// TIA Portal V19 export
FUNCTION_BLOCK "A0303_Sostegno_FB"   // FB102, LAD
// stored: MemoryReserve 100, SetENOAutomatically false
   VAR_INPUT
      AreaInterface : "AreaInterface";
      ZSI : "udt_ZoneSafetyInterface";
      DSI_Feed : "udt_DeviceSafetyInterface";
      DSI_Valve : "udt_DeviceSafetyInterface";
      DataIn : Struct
         OP_Work_PB : Bool;
         OP_Rest_PB : Bool;
         Pos0_Ls : Bool;
         Pos1_Ls : Bool;
         Pos2_Ls : Bool;
      END_STRUCT;
      CIn : Struct
         Manager : Struct
            EnableStopDoorOpeningReq : Bool;
            EnableStopInPhase : Bool;
            EnableStopProgrammed : Bool;
            Control_ON : Bool;
            CanMoveFreely : Bool;
            Phase : Struct
               VAI_A_LAVORO : Bool;
               VAI_A_RIPOSO : Bool;
            END_STRUCT;
            Ax : Struct
               Pos { ExternalVisible := 'False'; ExternalWritable := 'False'} : LReal;
            END_STRUCT;
            Paletti : Struct
               PosPaletto : Int;
               Pos1Collision : Bool;
               Pos2Collision : Bool;
            END_STRUCT;
         END_STRUCT;
         Navetta : Struct
            OutOfWorkspace : Bool;
         END_STRUCT;
         Trasporto : Struct
            OutOfWorkspace : Bool;
         END_STRUCT;
         CycleModeShortPiece : Bool;
      END_STRUCT;
      Config : Struct
         Ax : "Positioning_DOL_Machine_Config";
         V_1 : "ValveMachine_Config";
         V_2 : "ValveMachine_Config";
         DelayMissingCondition { ExternalAccessible := 'False'; ExternalVisible := 'False'; ExternalWritable := 'False'} : Time;
      END_STRUCT;
      HWID : Struct
         Ax_TEL1 : HW_SUBMODULE;
         Enc_IO : HW_SUBMODULE;
      END_STRUCT;
   END_VAR
   VAR_OUTPUT
      MachineInterface : "MachineInterface";
      COut : Struct
         Ax : "Positioning_DOL_Machine_COut";
         Paletto : Struct
            CtrlSafe : Bool;
            Standstill : Bool;
            Rest_CheckNext : Bool;
            Work_CheckNext : Bool;
            Pos : Int;
            RestPosition : Bool;
         END_STRUCT;
      END_STRUCT;
   END_VAR
   VAR_IN_OUT
      Par : Struct
         Ax : "Positioning_DOL_Machine_Par";
         Ax_Pers : "Positioning_DOL_Machine_Pers_Data";
         Enc : "PosFbk_RTN";
      END_STRUCT;
      Par_Mach : Struct
         RestPosition : LReal;
         ToleranceWindow : LReal;
         PosTimeout : Time;
      END_STRUCT;
   END_VAR
   VAR
      Alarm : Struct
         Ax { S7_SetPoint := 'True'} : "Positioning_DOL_Machine_Alr";
         V_1 : "ValveAlr";
         V_2 : "ValveAlr";
         Enc { S7_SetPoint := 'True'} : "PosFbk_Encoder_Alr";
         Missing_Pos0_Ls_ON { S7_SetPoint := 'True'} : Bool;
         Missing_Pos1_Ls_ON { S7_SetPoint := 'True'} : Bool;
         Missing_Pos2_Ls_ON { S7_SetPoint := 'True'} : Bool;
         LimitSwitch : Bool;
      END_STRUCT;
      Warning : Struct
         Ax { S7_SetPoint := 'True'} : "Positioning_DOL_Machine_Wng";
         V_1 { S7_SetPoint := 'True'} : "ValveMachine_Wng";
         V_2 { S7_SetPoint := 'True'} : "ValveMachine_Wng";
         V_Paletti { S7_SetPoint := 'True'} : "ValveMachine_Wng";
         MissingCnd : Struct
            OP_REST : Bool;   // Mancanza comando arresto
            OP_WORK : Bool;   // Mancanza consenso lavoro
            AxInRestPos : Bool;
         END_STRUCT;
      END_STRUCT;
      Ctrl : Struct
         Man : Struct
            OP_Vai_A_Lavoro : Bool;
            OP_Vai_A_Riposo : Bool;
         END_STRUCT;
         Aut : Struct
            OP_Vai_A_Lavoro : Bool;
            OP_Vai_A_Riposo : Bool;
         END_STRUCT;
         Pos0 : Bool;
         Pos1 : Bool;
         Pos2 : Bool;
         OP_Vai_A_Lavoro : Bool;
         OP_Vai_A_Riposo : Bool;
      END_STRUCT;
      Sts : Struct
         OP_Ax_CanMoveFreely : Bool;
         OP_CanMoveFreely : Bool;
         OP_Rest_Cnd : Bool;
         OP_Work_Cnd : Bool;
         InRestPos : Bool;
      END_STRUCT;
      HMI : Struct
         PbPreset : Bool;
         PresetValue : LReal;
      END_STRUCT;
      Ax { S7_SetPoint := 'True'} : "Positioning_DOL_Machine_FB";
      Enc : "PosFbk_SickAFM60";
      Enc_ITF : "PosFbk_ITF";
      V_1 { S7_SetPoint := 'True'} : "ValveMachine_FB";
      V_2 { S7_SetPoint := 'True'} : "ValveMachine_FB";
      AUX : Struct
         OP_Work_PB { ExternalAccessible := 'False'; ExternalVisible := 'False'; ExternalWritable := 'False'} : Bool;
         OP_Rest_PB { ExternalAccessible := 'False'; ExternalVisible := 'False'; ExternalWritable := 'False'} : Bool;
         OP_MoveToPos : Bool;
         PbPos0 : Bool;
         PbPos1 : Bool;
         PbPos2 : Bool;
      END_STRUCT;
      TON_MissingLsPos0 : IEC_TIMER;
      TON_MissingLsPos1 : IEC_TIMER;
      TON_MissingLsPos2 : IEC_TIMER;
      TON_OP_REST_MissingCnd : IEC_TIMER;
      TON_OP_WORK_MissingCnd : IEC_TIMER;
   END_VAR
   VAR_TEMP
      PE : Struct
         OP_Rest_PB : Bool;
         OP_Work_PB : Bool;
         PbPos0 : Bool;
         PbPos1 : Bool;
         PbPos2 : Bool;
      END_STRUCT;
      V1_Work_1 : Bool;
      V1_Work_2 : Bool;
      V1_Rest : Bool;
      V1_Rest_2 : Bool;
      V2_Work : Bool;
      V2_Rest_1 : Bool;
      V2_Rest_2 : Bool;
   END_VAR
   VAR_TEMP   // added for the SCL form of the ladder/FBD networks
      _w1 : Bool;
   END_VAR
BEGIN

REGION Network 1 (SCL): Reset allarmi
   IF #AreaInterface.RstAlarms THEN
       #Warning.MissingCnd.AxInRestPos:=FALSE;
   END_IF;
END_REGION

REGION Network 2: <+>
END_REGION

REGION Network 3: <+>
END_REGION

REGION Network 4: [Ax] - Operazione può muoversi liberamente perchè non sposta nessun BEAM
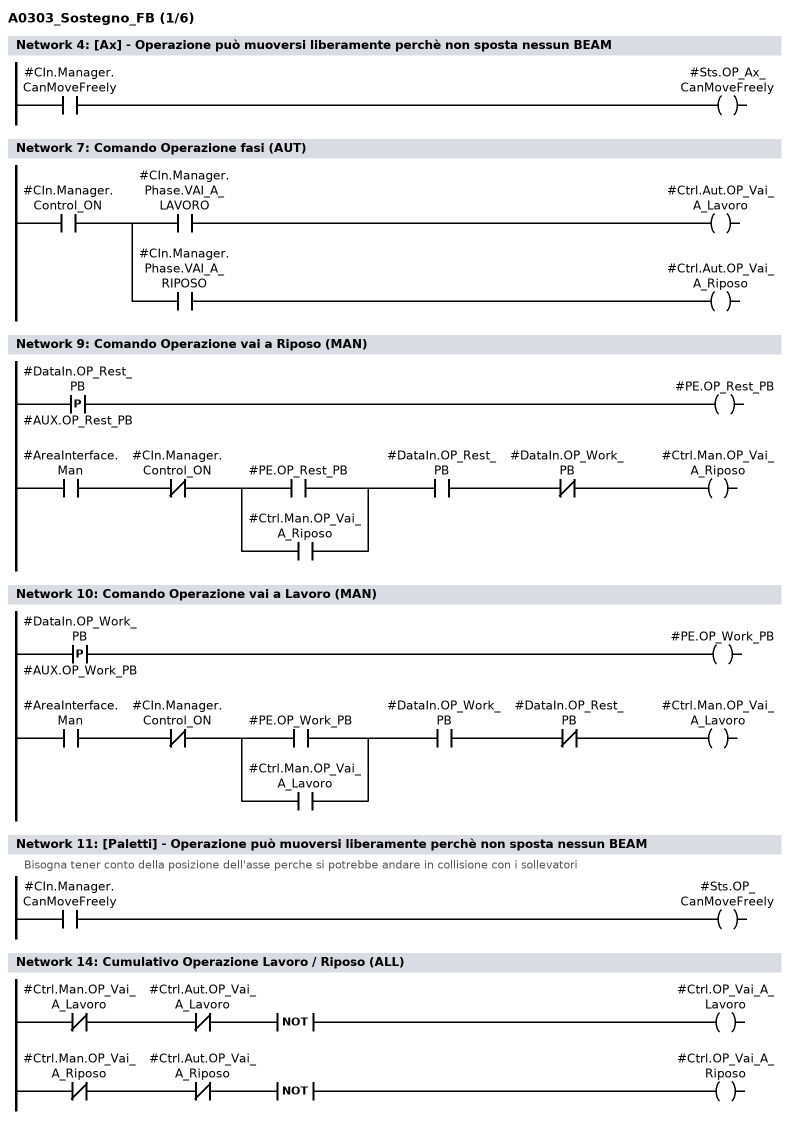
   RUNG wire#powerrail
      Contact( #CIn.Manager.CanMoveFreely )
      Coil( #Sts.OP_Ax_CanMoveFreely )
   END_RUNG
   // the same network as SCL:
   #Sts.OP_Ax_CanMoveFreely := #CIn.Manager.CanMoveFreely;
END_REGION

REGION Network 5: <+>
END_REGION

REGION Network 6: < OPERAZIONI AUTOMATICO >
END_REGION

REGION Network 7: Comando Operazione fasi (AUT)
   RUNG wire#powerrail
      Contact( #CIn.Manager.Control_ON )
      wire#w1
      Contact( #CIn.Manager.Phase.VAI_A_LAVORO )
      Coil( #Ctrl.Aut.OP_Vai_A_Lavoro )
   END_RUNG
   RUNG wire#w1
      Contact( #CIn.Manager.Phase.VAI_A_RIPOSO )
      Coil( #Ctrl.Aut.OP_Vai_A_Riposo )
   END_RUNG
   // the same network as SCL:
   #Ctrl.Aut.OP_Vai_A_Lavoro := #CIn.Manager.Control_ON AND #CIn.Manager.Phase.VAI_A_LAVORO;
   #Ctrl.Aut.OP_Vai_A_Riposo := #CIn.Manager.Control_ON AND #CIn.Manager.Phase.VAI_A_RIPOSO;
END_REGION

REGION Network 8: < OPERAZIONI MANUALI >
END_REGION

REGION Network 9: Comando Operazione vai a Riposo (MAN)
   RUNG wire#powerrail
      P_Contact(operand := #DataIn.OP_Rest_PB, bit := #AUX.OP_Rest_PB)
      Coil( #PE.OP_Rest_PB )
   END_RUNG
   RUNG wire#powerrail
      Contact( #AreaInterface.Man )
      I_Contact( #CIn.Manager.Control_ON )
      wire#w1
      Contact( #PE.OP_Rest_PB )
      wire#w2
      Contact( #DataIn.OP_Rest_PB )
      I_Contact( #DataIn.OP_Work_PB )
      Coil( #Ctrl.Man.OP_Vai_A_Riposo )
   END_RUNG
   RUNG wire#w1
      Contact( #Ctrl.Man.OP_Vai_A_Riposo )
   END_RUNG wire#w2
   // the same network as SCL:
   #_w1 := #DataIn.OP_Rest_PB AND NOT #AUX.OP_Rest_PB;   // rising edge of #DataIn.OP_Rest_PB
   #AUX.OP_Rest_PB := #DataIn.OP_Rest_PB;
   #PE.OP_Rest_PB := #_w1;
   #Ctrl.Man.OP_Vai_A_Riposo := #AreaInterface.Man AND NOT #CIn.Manager.Control_ON AND (#PE.OP_Rest_PB OR #Ctrl.Man.OP_Vai_A_Riposo) AND #DataIn.OP_Rest_PB AND NOT #DataIn.OP_Work_PB;
END_REGION

REGION Network 10: Comando Operazione vai a Lavoro (MAN)
   RUNG wire#powerrail
      P_Contact(operand := #DataIn.OP_Work_PB, bit := #AUX.OP_Work_PB)
      Coil( #PE.OP_Work_PB )
   END_RUNG
   RUNG wire#powerrail
      Contact( #AreaInterface.Man )
      I_Contact( #CIn.Manager.Control_ON )
      wire#w1
      Contact( #PE.OP_Work_PB )
      wire#w2
      Contact( #DataIn.OP_Work_PB )
      I_Contact( #DataIn.OP_Rest_PB )
      Coil( #Ctrl.Man.OP_Vai_A_Lavoro )
   END_RUNG
   RUNG wire#w1
      Contact( #Ctrl.Man.OP_Vai_A_Lavoro )
   END_RUNG wire#w2
   // the same network as SCL:
   #_w1 := #DataIn.OP_Work_PB AND NOT #AUX.OP_Work_PB;   // rising edge of #DataIn.OP_Work_PB
   #AUX.OP_Work_PB := #DataIn.OP_Work_PB;
   #PE.OP_Work_PB := #_w1;
   #Ctrl.Man.OP_Vai_A_Lavoro := #AreaInterface.Man AND NOT #CIn.Manager.Control_ON AND (#PE.OP_Work_PB OR #Ctrl.Man.OP_Vai_A_Lavoro) AND #DataIn.OP_Work_PB AND NOT #DataIn.OP_Rest_PB;
END_REGION

REGION Network 11: [Paletti] - Operazione può muoversi liberamente perchè non sposta nessun BEAM
   // Bisogna tener conto della posizione dell'asse perche si potrebbe andare in collisione con i sollevatori
   RUNG wire#powerrail
      Contact( #CIn.Manager.CanMoveFreely )
      Coil( #Sts.OP_CanMoveFreely )
   END_RUNG
   // the same network as SCL:
   #Sts.OP_CanMoveFreely := #CIn.Manager.CanMoveFreely;
END_REGION

REGION Network 12: <+>
END_REGION

REGION Network 13: < CUMULATIVO OPERAZIONI >
END_REGION

REGION Network 14: Cumulativo Operazione Lavoro / Riposo (ALL)
   RUNG wire#powerrail
      I_Contact( #Ctrl.Man.OP_Vai_A_Lavoro )
      I_Contact( #Ctrl.Aut.OP_Vai_A_Lavoro )
      Not()
      Coil( #Ctrl.OP_Vai_A_Lavoro )
   END_RUNG
   RUNG wire#powerrail
      I_Contact( #Ctrl.Man.OP_Vai_A_Riposo )
      I_Contact( #Ctrl.Aut.OP_Vai_A_Riposo )
      Not()
      Coil( #Ctrl.OP_Vai_A_Riposo )
   END_RUNG
   // the same network as SCL:
   #Ctrl.OP_Vai_A_Lavoro := NOT (NOT #Ctrl.Man.OP_Vai_A_Lavoro AND NOT #Ctrl.Aut.OP_Vai_A_Lavoro);
   #Ctrl.OP_Vai_A_Riposo := NOT (NOT #Ctrl.Man.OP_Vai_A_Riposo AND NOT #Ctrl.Aut.OP_Vai_A_Riposo);
END_REGION

REGION Network 15: < CONDIZIONI MOVIMENTO >
END_REGION

REGION Network 16: Condizioni movimento Operazione a Lavoro / Riposo
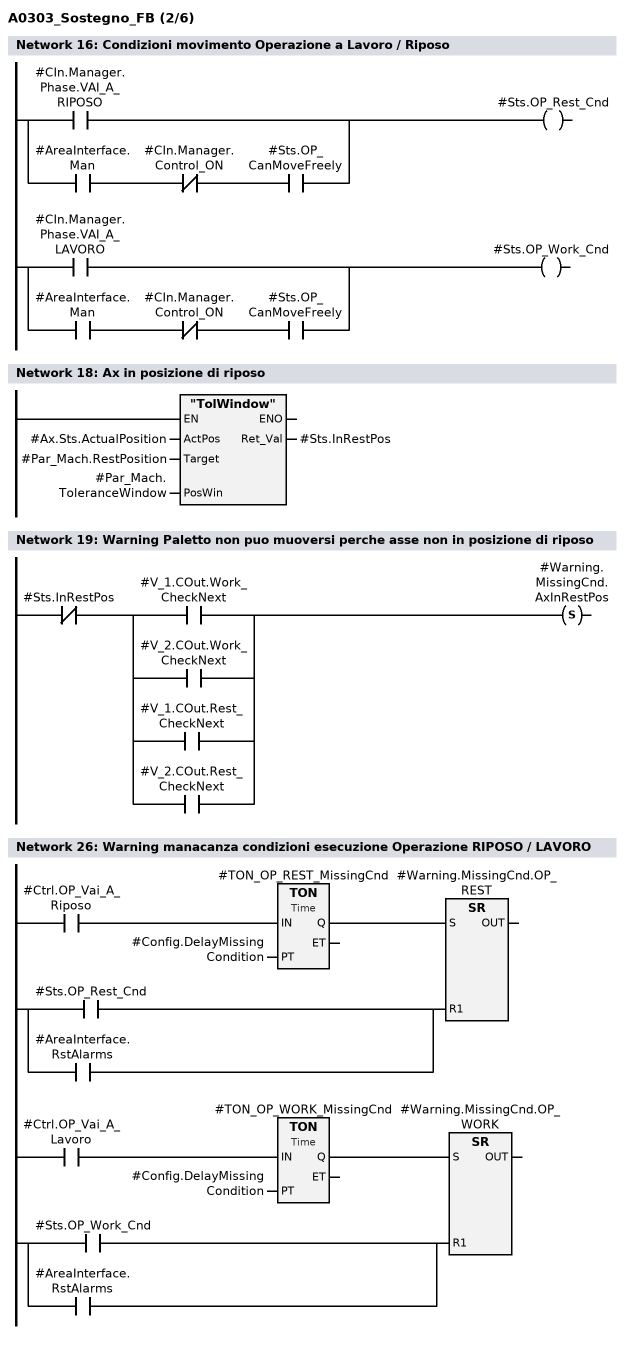
   RUNG wire#powerrail
      Contact( #CIn.Manager.Phase.VAI_A_RIPOSO )
      wire#w1
      Coil( #Sts.OP_Rest_Cnd )
   END_RUNG
   RUNG wire#powerrail
      Contact( #AreaInterface.Man )
      I_Contact( #CIn.Manager.Control_ON )
      Contact( #Sts.OP_CanMoveFreely )
   END_RUNG wire#w1
   RUNG wire#powerrail
      Contact( #CIn.Manager.Phase.VAI_A_LAVORO )
      wire#w2
      Coil( #Sts.OP_Work_Cnd )
   END_RUNG
   RUNG wire#powerrail
      Contact( #AreaInterface.Man )
      I_Contact( #CIn.Manager.Control_ON )
      Contact( #Sts.OP_CanMoveFreely )
   END_RUNG wire#w2
   // the same network as SCL:
   #Sts.OP_Rest_Cnd := #CIn.Manager.Phase.VAI_A_RIPOSO OR (#AreaInterface.Man AND NOT #CIn.Manager.Control_ON AND #Sts.OP_CanMoveFreely);
   #Sts.OP_Work_Cnd := #CIn.Manager.Phase.VAI_A_LAVORO OR (#AreaInterface.Man AND NOT #CIn.Manager.Control_ON AND #Sts.OP_CanMoveFreely);
END_REGION

REGION Network 17: <+>
END_REGION

REGION Network 18: Ax in posizione di riposo
   RUNG wire#powerrail
      "TolWindow"(ActPos := #Ax.Sts.ActualPosition, Target := #Par_Mach.RestPosition, PosWin := #Par_Mach.ToleranceWindow, Ret_Val => #Sts.InRestPos)
   END_RUNG
   // the same network as SCL:
   #Sts.InRestPos := "TolWindow"(ActPos := #Ax.Sts.ActualPosition,
                           Target := #Par_Mach.RestPosition,
                           PosWin := #Par_Mach.ToleranceWindow);
END_REGION

REGION Network 19: Warning Paletto non puo muoversi perche asse non in posizione di riposo
   RUNG wire#powerrail
      I_Contact( #Sts.InRestPos )
      wire#w1
      Contact( #V_1.COut.Work_CheckNext )
      wire#w2
      S_Coil( #Warning.MissingCnd.AxInRestPos )
   END_RUNG
   RUNG wire#w1
      Contact( #V_2.COut.Work_CheckNext )
   END_RUNG wire#w2
   RUNG wire#w1
      Contact( #V_1.COut.Rest_CheckNext )
   END_RUNG wire#w2
   RUNG wire#w1
      Contact( #V_2.COut.Rest_CheckNext )
   END_RUNG wire#w2
   // the same network as SCL:
   IF NOT #Sts.InRestPos AND (#V_1.COut.Work_CheckNext OR #V_2.COut.Work_CheckNext OR #V_1.COut.Rest_CheckNext OR #V_2.COut.Rest_CheckNext) THEN
       #Warning.MissingCnd.AxInRestPos := TRUE;
   END_IF;
END_REGION

REGION Network 20: <+>
END_REGION

REGION Network 21 (SCL): CIn Abilitazioni Manager
   //Stop Door Opening Request
   #Ax.CIn.Manager.EnableStopDoorOpeningReq :=
   #V_1.Cin.Manager.EnableStopDoorOpeningReq := #V_2.Cin.Manager.EnableStopDoorOpeningReq := #CIn.Manager.EnableStopDoorOpeningReq;

   //Stop In Phase
   #Ax.CIn.Manager.EnableStopInPhase := 
   #V_1.Cin.Manager.EnableStopInPhase := #V_2.Cin.Manager.EnableStopInPhase := #CIn.Manager.EnableStopInPhase;

   //Stop Programmed
   #Ax.CIn.Manager.EnableStopProgrammed := 
   #V_1.Cin.Manager.EnableStopProgrammed := #V_2.Cin.Manager.EnableStopProgrammed :=#CIn.Manager.EnableStopProgrammed;
END_REGION

REGION Network 22: <+>
END_REGION

REGION Network 23: <+>
END_REGION

REGION Network 24: <<<MANAGER >>>
END_REGION

REGION Network 25 (SCL): Cin Manager (Esecuzione sequenza comandi)
   //CTRL ON
   #Ax.CIn.Manager.Control_ON :=#V_1.Cin.Manager.Control_ON :=#V_2.Cin.Manager.Control_ON := #Ctrl.OP_Vai_A_Lavoro OR #Ctrl.OP_Vai_A_Riposo;


   IF #Ctrl.OP_Vai_A_Lavoro AND #Sts.OP_Work_Cnd THEN


       IF #CIn.Manager.Paletti.PosPaletto = 1 THEN
           #Ctrl.Pos1 := NOT #DataIn.Pos1_Ls;
       ELSIF #CIn.Manager.Paletti.PosPaletto = 2 THEN
           #Ctrl.Pos2 := NOT #DataIn.Pos2_Ls;
       END_IF;

       #Ax.CIn.Manager.Speed := 100;
       #Ax.CIn.Manager.MoveToPos := #CIn.Manager.Paletti.PosPaletto = #COut.Paletto.Pos;
       #Ax.CIn.Manager.Pos := #CIn.Manager.Ax.Pos;




   ELSIF #Ctrl.OP_Vai_A_Riposo AND #Sts.OP_Rest_Cnd THEN



       IF NOT #CIn.CycleModeShortPiece THEN

           #Ax.CIn.Manager.Speed := 100;
           #Ax.CIn.Manager.MoveToPos := #CIn.Manager.Paletti.PosPaletto = #COut.Paletto.Pos;
           #Ax.CIn.Manager.Pos := #Par_Mach.RestPosition;

           IF #Sts.InRestPos THEN
               #Ctrl.Pos0 := NOT #DataIn.Pos0_Ls;
           END_IF;

       ELSE

           #Ctrl.Pos0 := NOT #DataIn.Pos0_Ls;


       END_IF;

   ELSE
       #Ctrl.Pos0 := #Ctrl.Pos1 := #Ctrl.Pos2 :=  #Ax.CIn.Manager.MoveToPos:= FALSE;


   END_IF;
END_REGION

REGION Network 26: Warning manacanza condizioni esecuzione Operazione RIPOSO / LAVORO
   RUNG wire#powerrail
      Contact( #Ctrl.OP_Vai_A_Riposo )
      { S7_Templates := "time_type := Time" } #TON_OP_REST_MissingCnd.TON(pt := #Config.DelayMissingCondition, et =>)
      S_SR(operand := #Warning.MissingCnd.OP_REST, r1 := wire#w1)
   END_RUNG
   RUNG wire#powerrail
      Contact( #Sts.OP_Rest_Cnd )
   END_RUNG wire#w1
   RUNG wire#powerrail
      Contact( #AreaInterface.RstAlarms )
   END_RUNG wire#w1
   RUNG wire#powerrail
      Contact( #Ctrl.OP_Vai_A_Lavoro )
      { S7_Templates := "time_type := Time" } #TON_OP_WORK_MissingCnd.TON(pt := #Config.DelayMissingCondition, et =>)
      S_SR(operand := #Warning.MissingCnd.OP_WORK, r1 := wire#w2)
   END_RUNG
   RUNG wire#powerrail
      Contact( #Sts.OP_Work_Cnd )
   END_RUNG wire#w2
   RUNG wire#powerrail
      Contact( #AreaInterface.RstAlarms )
   END_RUNG wire#w2
   // the same network as SCL:
   #TON_OP_REST_MissingCnd.TON(IN := #Ctrl.OP_Vai_A_Riposo, PT := #Config.DelayMissingCondition);
   IF #TON_OP_REST_MissingCnd.Q THEN
       #Warning.MissingCnd.OP_REST := TRUE;   // SR flip-flop
   END_IF;
   IF #Sts.OP_Rest_Cnd OR #AreaInterface.RstAlarms THEN #Warning.MissingCnd.OP_REST := FALSE; END_IF;
   #TON_OP_WORK_MissingCnd.TON(IN := #Ctrl.OP_Vai_A_Lavoro, PT := #Config.DelayMissingCondition);
   IF #TON_OP_WORK_MissingCnd.Q THEN
       #Warning.MissingCnd.OP_WORK := TRUE;   // SR flip-flop
   END_IF;
   IF #Sts.OP_Work_Cnd OR #AreaInterface.RstAlarms THEN #Warning.MissingCnd.OP_WORK := FALSE; END_IF;
END_REGION

REGION Network 27: <+>
END_REGION

REGION Network 28: <<< ASSE Y >>>
END_REGION

REGION Network 29: [Ax] - Cin Ext Enable
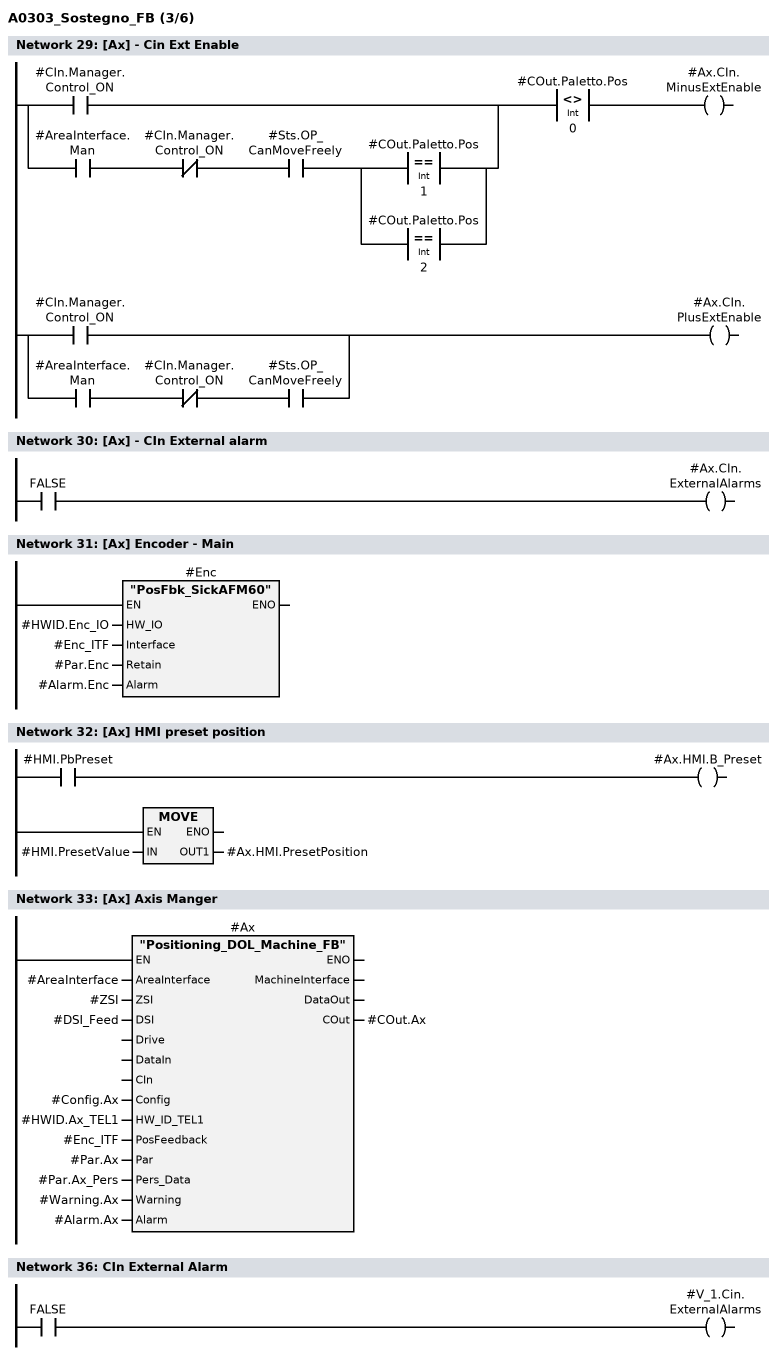
   RUNG wire#powerrail
      Contact( #CIn.Manager.Control_ON )
      wire#w1
      { S7_Templates := "SrcType := Int" } NE_Contact(in1 := #COut.Paletto.Pos, in2 := 0)
      Coil( #Ax.CIn.MinusExtEnable )
   END_RUNG
   RUNG wire#powerrail
      Contact( #AreaInterface.Man )
      I_Contact( #CIn.Manager.Control_ON )
      Contact( #Sts.OP_CanMoveFreely )
      wire#w2
      { S7_Templates := "SrcType := Int" } EQ_Contact(in1 := #COut.Paletto.Pos, in2 := 1)
   END_RUNG wire#w1
   RUNG wire#w2
      { S7_Templates := "SrcType := Int" } EQ_Contact(in1 := #COut.Paletto.Pos, in2 := 2)
   END_RUNG wire#w1
   RUNG wire#powerrail
      Contact( #CIn.Manager.Control_ON )
      wire#w3
      Coil( #Ax.CIn.PlusExtEnable )
   END_RUNG
   RUNG wire#powerrail
      Contact( #AreaInterface.Man )
      I_Contact( #CIn.Manager.Control_ON )
      Contact( #Sts.OP_CanMoveFreely )
   END_RUNG wire#w3
   // the same network as SCL:
   #Ax.CIn.MinusExtEnable := (#CIn.Manager.Control_ON OR (#AreaInterface.Man AND NOT #CIn.Manager.Control_ON AND #Sts.OP_CanMoveFreely AND ((#COut.Paletto.Pos = 1) OR (#COut.Paletto.Pos = 2)))) AND (#COut.Paletto.Pos <> 0);
   #Ax.CIn.PlusExtEnable := #CIn.Manager.Control_ON OR (#AreaInterface.Man AND NOT #CIn.Manager.Control_ON AND #Sts.OP_CanMoveFreely);
END_REGION

REGION Network 30: [Ax] - CIn External alarm
   RUNG wire#powerrail
      Contact( FALSE )
      Coil( #Ax.CIn.ExternalAlarms )
   END_RUNG
   // the same network as SCL:
   #Ax.CIn.ExternalAlarms := FALSE;
END_REGION

REGION Network 31: [Ax] Encoder - Main
   RUNG wire#powerrail
      #Enc(HW_IO := #HWID.Enc_IO, Interface := #Enc_ITF, Retain := #Par.Enc, Alarm := #Alarm.Enc)
   END_RUNG
   // the same network as SCL:
   #Enc(HW_IO := #HWID.Enc_IO, Interface := #Enc_ITF, Retain := #Par.Enc, Alarm := #Alarm.Enc);   // "PosFbk_SickAFM60"
END_REGION

REGION Network 32: [Ax] HMI preset position
   RUNG wire#powerrail
      Contact( #HMI.PbPreset )
      Coil( #Ax.HMI.B_Preset )
   END_RUNG
   RUNG wire#powerrail
      Move(in := #HMI.PresetValue, out1 => #Ax.HMI.PresetPosition)
   END_RUNG
   // the same network as SCL:
   #Ax.HMI.B_Preset := #HMI.PbPreset;
   #Ax.HMI.PresetPosition := #HMI.PresetValue;
END_REGION

REGION Network 33: [Ax] Axis Manger
   RUNG wire#powerrail
      #Ax(AreaInterface := #AreaInterface, ZSI := #ZSI, DSI := #DSI_Feed, Drive :=, DataIn :=, CIn :=, Config := #Config.Ax, HW_ID_TEL1 := #HWID.Ax_TEL1, PosFeedback := #Enc_ITF, Par := #Par.Ax, Pers_Data := #Par.Ax_Pers, Warning := #Warning.Ax, Alarm := #Alarm.Ax, MachineInterface =>, DataOut =>, COut => #COut.Ax)
   END_RUNG
   // the same network as SCL:
   #Ax(AreaInterface := #AreaInterface,   // "Positioning_DOL_Machine_FB"
       ZSI := #ZSI,
       DSI := #DSI_Feed,
       Config := #Config.Ax,
       HW_ID_TEL1 := #HWID.Ax_TEL1,
       PosFeedback := #Enc_ITF,
       Par := #Par.Ax,
       Pers_Data := #Par.Ax_Pers,
       Warning := #Warning.Ax,
       Alarm := #Alarm.Ax,
       COut => #COut.Ax);
END_REGION

REGION Network 35: <<< VALVE 1>>>
END_REGION

REGION Network 36: CIn External Alarm
   RUNG wire#powerrail
      Contact( FALSE )
      Coil( #V_1.Cin.ExternalAlarms )
   END_RUNG
   // the same network as SCL:
   #V_1.Cin.ExternalAlarms := FALSE;
END_REGION

REGION Network 37: CIn External Enable
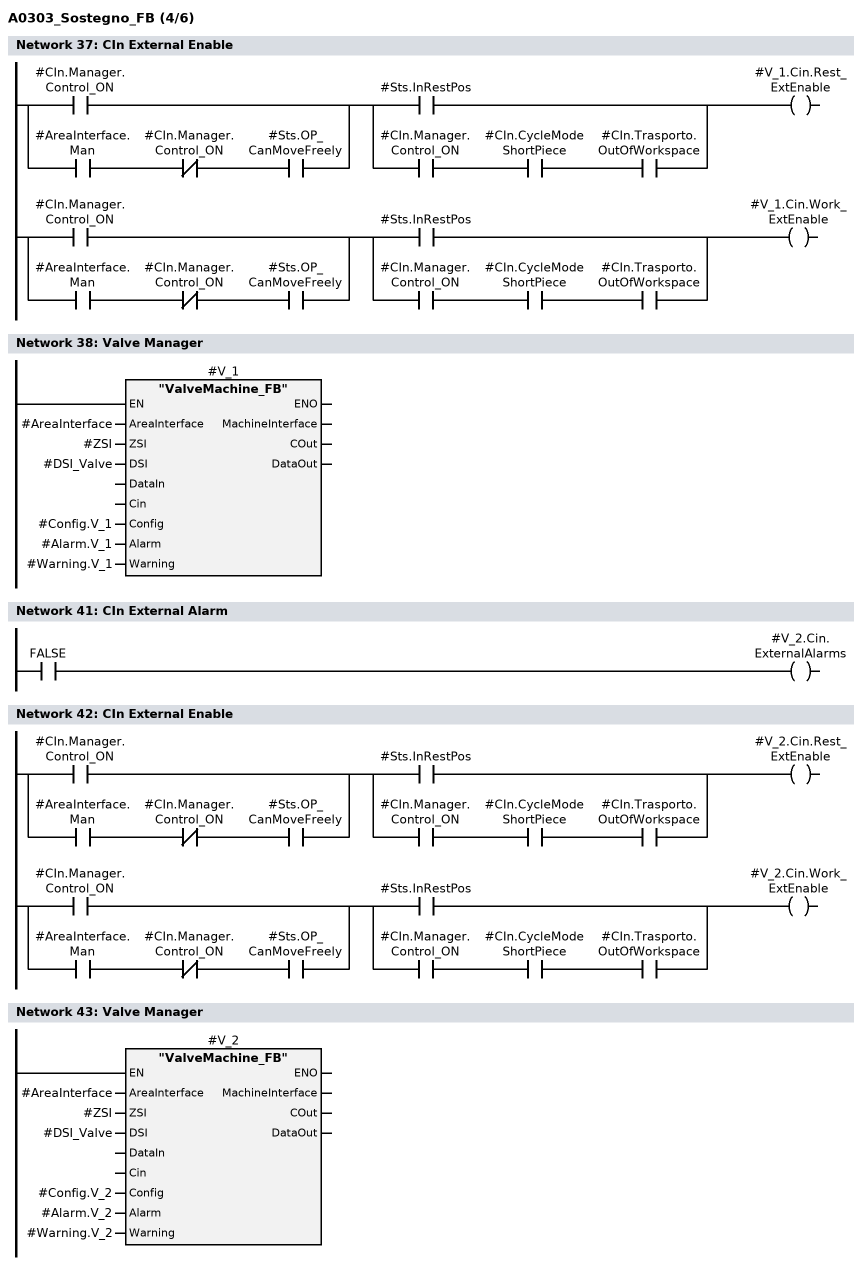
   RUNG wire#powerrail
      Contact( #CIn.Manager.Control_ON )
      wire#w1
      Contact( #Sts.InRestPos )
      wire#w2
      Coil( #V_1.Cin.Rest_ExtEnable )
   END_RUNG
   RUNG wire#powerrail
      Contact( #AreaInterface.Man )
      I_Contact( #CIn.Manager.Control_ON )
      Contact( #Sts.OP_CanMoveFreely )
   END_RUNG wire#w1
   RUNG wire#w1
      Contact( #CIn.Manager.Control_ON )
      Contact( #CIn.CycleModeShortPiece )
      Contact( #CIn.Trasporto.OutOfWorkspace )
   END_RUNG wire#w2
   RUNG wire#powerrail
      Contact( #CIn.Manager.Control_ON )
      wire#w3
      Contact( #Sts.InRestPos )
      wire#w4
      Coil( #V_1.Cin.Work_ExtEnable )
   END_RUNG
   RUNG wire#powerrail
      Contact( #AreaInterface.Man )
      I_Contact( #CIn.Manager.Control_ON )
      Contact( #Sts.OP_CanMoveFreely )
   END_RUNG wire#w3
   RUNG wire#w3
      Contact( #CIn.Manager.Control_ON )
      Contact( #CIn.CycleModeShortPiece )
      Contact( #CIn.Trasporto.OutOfWorkspace )
   END_RUNG wire#w4
   // the same network as SCL:
   #V_1.Cin.Rest_ExtEnable := (#CIn.Manager.Control_ON OR (#AreaInterface.Man AND NOT #CIn.Manager.Control_ON AND #Sts.OP_CanMoveFreely)) AND (#Sts.InRestPos OR (#CIn.Manager.Control_ON AND #CIn.CycleModeShortPiece AND #CIn.Trasporto.OutOfWorkspace));
   #V_1.Cin.Work_ExtEnable := (#CIn.Manager.Control_ON OR (#AreaInterface.Man AND NOT #CIn.Manager.Control_ON AND #Sts.OP_CanMoveFreely)) AND (#Sts.InRestPos OR (#CIn.Manager.Control_ON AND #CIn.CycleModeShortPiece AND #CIn.Trasporto.OutOfWorkspace));
END_REGION

REGION Network 38: Valve Manager
   RUNG wire#powerrail
      #V_1(AreaInterface := #AreaInterface, ZSI := #ZSI, DSI := #DSI_Valve, DataIn :=, Cin :=, Config := #Config.V_1, Alarm := #Alarm.V_1, Warning := #Warning.V_1, MachineInterface =>, COut =>, DataOut =>)
   END_RUNG
   // the same network as SCL:
   #V_1(AreaInterface := #AreaInterface,   // "ValveMachine_FB"
        ZSI := #ZSI,
        DSI := #DSI_Valve,
        Config := #Config.V_1,
        Alarm := #Alarm.V_1,
        Warning := #Warning.V_1);
END_REGION

REGION Network 40: <<<VALVE 2>>>
END_REGION

REGION Network 41: CIn External Alarm
   RUNG wire#powerrail
      Contact( FALSE )
      Coil( #V_2.Cin.ExternalAlarms )
   END_RUNG
   // the same network as SCL:
   #V_2.Cin.ExternalAlarms := FALSE;
END_REGION

REGION Network 42: CIn External Enable
   RUNG wire#powerrail
      Contact( #CIn.Manager.Control_ON )
      wire#w1
      Contact( #Sts.InRestPos )
      wire#w2
      Coil( #V_2.Cin.Rest_ExtEnable )
   END_RUNG
   RUNG wire#powerrail
      Contact( #AreaInterface.Man )
      I_Contact( #CIn.Manager.Control_ON )
      Contact( #Sts.OP_CanMoveFreely )
   END_RUNG wire#w1
   RUNG wire#w1
      Contact( #CIn.Manager.Control_ON )
      Contact( #CIn.CycleModeShortPiece )
      Contact( #CIn.Trasporto.OutOfWorkspace )
   END_RUNG wire#w2
   RUNG wire#powerrail
      Contact( #CIn.Manager.Control_ON )
      wire#w3
      Contact( #Sts.InRestPos )
      wire#w4
      Coil( #V_2.Cin.Work_ExtEnable )
   END_RUNG
   RUNG wire#powerrail
      Contact( #AreaInterface.Man )
      I_Contact( #CIn.Manager.Control_ON )
      Contact( #Sts.OP_CanMoveFreely )
   END_RUNG wire#w3
   RUNG wire#w3
      Contact( #CIn.Manager.Control_ON )
      Contact( #CIn.CycleModeShortPiece )
      Contact( #CIn.Trasporto.OutOfWorkspace )
   END_RUNG wire#w4
   // the same network as SCL:
   #V_2.Cin.Rest_ExtEnable := (#CIn.Manager.Control_ON OR (#AreaInterface.Man AND NOT #CIn.Manager.Control_ON AND #Sts.OP_CanMoveFreely)) AND (#Sts.InRestPos OR (#CIn.Manager.Control_ON AND #CIn.CycleModeShortPiece AND #CIn.Trasporto.OutOfWorkspace));
   #V_2.Cin.Work_ExtEnable := (#CIn.Manager.Control_ON OR (#AreaInterface.Man AND NOT #CIn.Manager.Control_ON AND #Sts.OP_CanMoveFreely)) AND (#Sts.InRestPos OR (#CIn.Manager.Control_ON AND #CIn.CycleModeShortPiece AND #CIn.Trasporto.OutOfWorkspace));
END_REGION

REGION Network 43: Valve Manager
   RUNG wire#powerrail
      #V_2(AreaInterface := #AreaInterface, ZSI := #ZSI, DSI := #DSI_Valve, DataIn :=, Cin :=, Config := #Config.V_2, Alarm := #Alarm.V_2, Warning := #Warning.V_2, MachineInterface =>, COut =>, DataOut =>)
   END_RUNG
   // the same network as SCL:
   #V_2(AreaInterface := #AreaInterface,   // "ValveMachine_FB"
        ZSI := #ZSI,
        DSI := #DSI_Valve,
        Config := #Config.V_2,
        Alarm := #Alarm.V_2,
        Warning := #Warning.V_2);
END_REGION

REGION Network 45: <<< VALVE CUMULATIVE >>>
END_REGION

REGION Network 46: [Paletti] - Alarm Ls
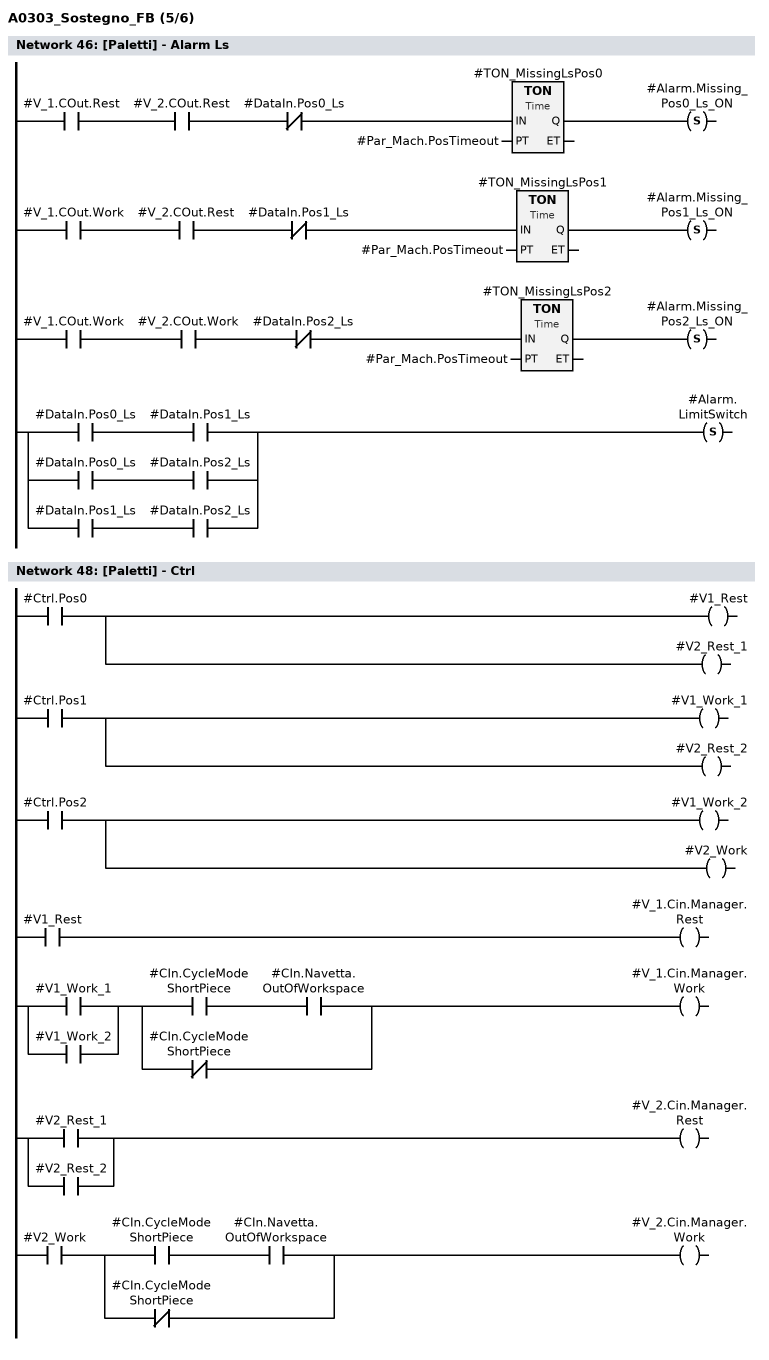
   RUNG wire#powerrail
      Contact( #V_1.COut.Rest )
      Contact( #V_2.COut.Rest )
      I_Contact( #DataIn.Pos0_Ls )
      { S7_Templates := "time_type := Time" } #TON_MissingLsPos0.TON(pt := #Par_Mach.PosTimeout, et =>)
      S_Coil( #Alarm.Missing_Pos0_Ls_ON )
   END_RUNG
   RUNG wire#powerrail
      Contact( #V_1.COut.Work )
      Contact( #V_2.COut.Rest )
      I_Contact( #DataIn.Pos1_Ls )
      { S7_Templates := "time_type := Time" } #TON_MissingLsPos1.TON(pt := #Par_Mach.PosTimeout, et =>)
      S_Coil( #Alarm.Missing_Pos1_Ls_ON )
   END_RUNG
   RUNG wire#powerrail
      Contact( #V_1.COut.Work )
      Contact( #V_2.COut.Work )
      I_Contact( #DataIn.Pos2_Ls )
      { S7_Templates := "time_type := Time" } #TON_MissingLsPos2.TON(pt := #Par_Mach.PosTimeout, et =>)
      S_Coil( #Alarm.Missing_Pos2_Ls_ON )
   END_RUNG
   RUNG wire#powerrail
      Contact( #DataIn.Pos0_Ls )
      Contact( #DataIn.Pos1_Ls )
      wire#w1
      S_Coil( #Alarm.LimitSwitch )
   END_RUNG
   RUNG wire#powerrail
      Contact( #DataIn.Pos0_Ls )
      Contact( #DataIn.Pos2_Ls )
   END_RUNG wire#w1
   RUNG wire#powerrail
      Contact( #DataIn.Pos1_Ls )
      Contact( #DataIn.Pos2_Ls )
   END_RUNG wire#w1
   // the same network as SCL:
   #TON_MissingLsPos0.TON(IN := #V_1.COut.Rest AND #V_2.COut.Rest AND NOT #DataIn.Pos0_Ls,
                          PT := #Par_Mach.PosTimeout);
   IF #TON_MissingLsPos0.Q THEN #Alarm.Missing_Pos0_Ls_ON := TRUE; END_IF;
   #TON_MissingLsPos1.TON(IN := #V_1.COut.Work AND #V_2.COut.Rest AND NOT #DataIn.Pos1_Ls,
                          PT := #Par_Mach.PosTimeout);
   IF #TON_MissingLsPos1.Q THEN #Alarm.Missing_Pos1_Ls_ON := TRUE; END_IF;
   #TON_MissingLsPos2.TON(IN := #V_1.COut.Work AND #V_2.COut.Work AND NOT #DataIn.Pos2_Ls,
                          PT := #Par_Mach.PosTimeout);
   IF #TON_MissingLsPos2.Q THEN #Alarm.Missing_Pos2_Ls_ON := TRUE; END_IF;
   IF (#DataIn.Pos0_Ls AND #DataIn.Pos1_Ls) OR (#DataIn.Pos0_Ls AND #DataIn.Pos2_Ls) OR (#DataIn.Pos1_Ls AND #DataIn.Pos2_Ls) THEN
       #Alarm.LimitSwitch := TRUE;
   END_IF;
END_REGION

REGION Network 47 (SCL): [Paletti] Warning
   #Warning.V_Paletti.NotAutReady:= #Warning.V_1.NotAutReady OR #Warning.V_2.NotAutReady;
   #Warning.V_Paletti.PressureRunning_Timeout := #Warning.V_1.PressureRunning_Timeout OR #Warning.V_2.PressureRunning_Timeout;
   #Warning.V_Paletti.Rest_MissingExtEnable := #Warning.V_1.Rest_MissingExtEnable OR #Warning.V_2.Rest_MissingExtEnable;
   #Warning.V_Paletti.Work_MissingExtEnable := #Warning.V_1.Work_MissingExtEnable OR #Warning.V_2.Work_MissingExtEnable;
   #Warning.V_Paletti.Missing_Rest_Ls_ON[1] := #Warning.V_1.Missing_Rest_Ls_ON[1] OR #Warning.V_2.Missing_Rest_Ls_ON[1];
   #Warning.V_Paletti.Missing_Work_Ls_ON[1] := #Warning.V_1.Missing_Work_Ls_ON[1] OR #Warning.V_2.Missing_Work_Ls_ON[1];
END_REGION

REGION Network 48: [Paletti] - Ctrl
   RUNG wire#powerrail
      Contact( #Ctrl.Pos0 )
      wire#w1
      Coil( #V1_Rest )
   END_RUNG
   RUNG wire#w1
      Coil( #V2_Rest_1 )
   END_RUNG
   RUNG wire#powerrail
      Contact( #Ctrl.Pos1 )
      wire#w2
      Coil( #V1_Work_1 )
   END_RUNG
   RUNG wire#w2
      Coil( #V2_Rest_2 )
   END_RUNG
   RUNG wire#powerrail
      Contact( #Ctrl.Pos2 )
      wire#w3
      Coil( #V1_Work_2 )
   END_RUNG
   RUNG wire#w3
      Coil( #V2_Work )
   END_RUNG
   RUNG wire#powerrail
      Contact( #V1_Rest )
      Coil( #V_1.Cin.Manager.Rest )
   END_RUNG
   RUNG wire#powerrail
      Contact( #V1_Work_1 )
      wire#w4
      Contact( #CIn.CycleModeShortPiece )
      Contact( #CIn.Navetta.OutOfWorkspace )
      wire#w5
      Coil( #V_1.Cin.Manager.Work )
   END_RUNG
   RUNG wire#powerrail
      Contact( #V1_Work_2 )
   END_RUNG wire#w4
   RUNG wire#w4
      I_Contact( #CIn.CycleModeShortPiece )
   END_RUNG wire#w5
   RUNG wire#powerrail
      Contact( #V2_Rest_1 )
      wire#w6
      Coil( #V_2.Cin.Manager.Rest )
   END_RUNG
   RUNG wire#powerrail
      Contact( #V2_Rest_2 )
   END_RUNG wire#w6
   RUNG wire#powerrail
      Contact( #V2_Work )
      wire#w7
      Contact( #CIn.CycleModeShortPiece )
      Contact( #CIn.Navetta.OutOfWorkspace )
      wire#w8
      Coil( #V_2.Cin.Manager.Work )
   END_RUNG
   RUNG wire#w7
      I_Contact( #CIn.CycleModeShortPiece )
   END_RUNG wire#w8
   // the same network as SCL:
   #V1_Rest := #Ctrl.Pos0;
   #V2_Rest_1 := #Ctrl.Pos0;
   #V1_Work_1 := #Ctrl.Pos1;
   #V2_Rest_2 := #Ctrl.Pos1;
   #V1_Work_2 := #Ctrl.Pos2;
   #V2_Work := #Ctrl.Pos2;
   #V_1.Cin.Manager.Rest := #V1_Rest;
   #V_1.Cin.Manager.Work := (#V1_Work_1 OR #V1_Work_2) AND ((#CIn.CycleModeShortPiece AND #CIn.Navetta.OutOfWorkspace) OR NOT #CIn.CycleModeShortPiece);
   #V_2.Cin.Manager.Rest := #V2_Rest_1 OR #V2_Rest_2;
   #V_2.Cin.Manager.Work := #V2_Work AND ((#CIn.CycleModeShortPiece AND #CIn.Navetta.OutOfWorkspace) OR NOT #CIn.CycleModeShortPiece);
END_REGION

REGION Network 49: [Paletti] - COut
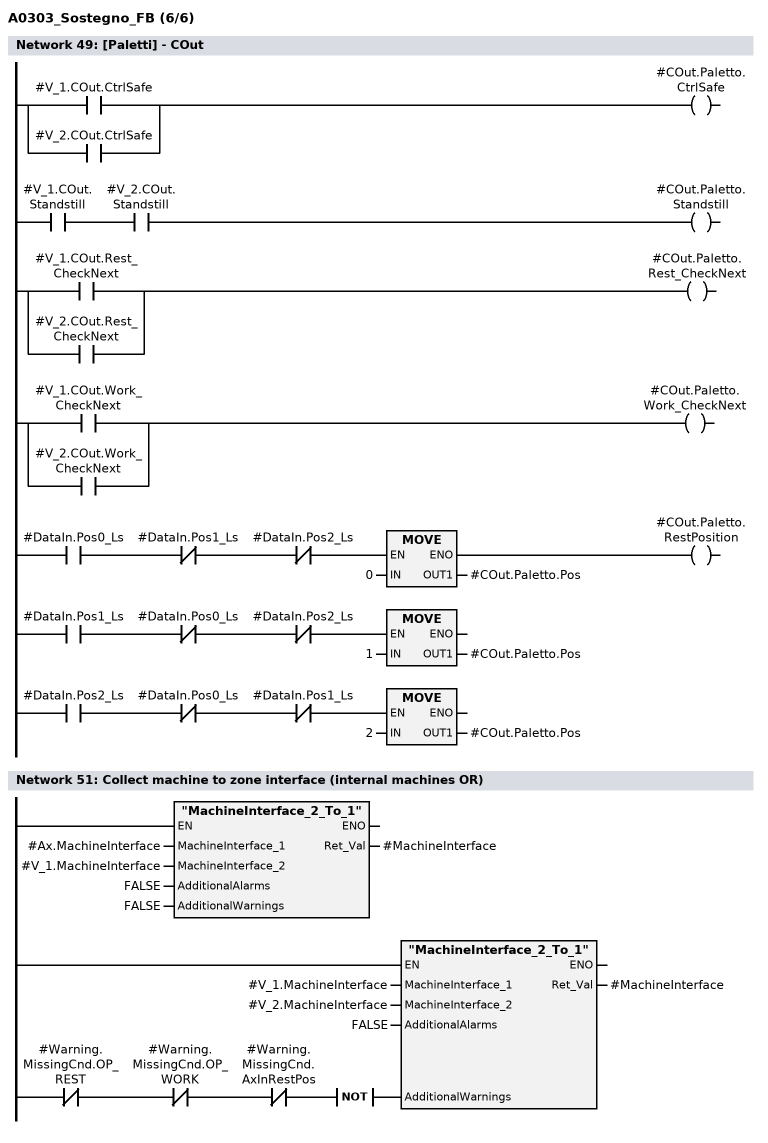
   RUNG wire#powerrail
      Contact( #V_1.COut.CtrlSafe )
      wire#w1
      Coil( #COut.Paletto.CtrlSafe )
   END_RUNG
   RUNG wire#powerrail
      Contact( #V_2.COut.CtrlSafe )
   END_RUNG wire#w1
   RUNG wire#powerrail
      Contact( #V_1.COut.Standstill )
      Contact( #V_2.COut.Standstill )
      Coil( #COut.Paletto.Standstill )
   END_RUNG
   RUNG wire#powerrail
      Contact( #V_1.COut.Rest_CheckNext )
      wire#w2
      Coil( #COut.Paletto.Rest_CheckNext )
   END_RUNG
   RUNG wire#powerrail
      Contact( #V_2.COut.Rest_CheckNext )
   END_RUNG wire#w2
   RUNG wire#powerrail
      Contact( #V_1.COut.Work_CheckNext )
      wire#w3
      Coil( #COut.Paletto.Work_CheckNext )
   END_RUNG
   RUNG wire#powerrail
      Contact( #V_2.COut.Work_CheckNext )
   END_RUNG wire#w3
   RUNG wire#powerrail
      Contact( #DataIn.Pos0_Ls )
      I_Contact( #DataIn.Pos1_Ls )
      I_Contact( #DataIn.Pos2_Ls )
      Move(in := 0, out1 => #COut.Paletto.Pos)
      Coil( #COut.Paletto.RestPosition )
   END_RUNG
   RUNG wire#powerrail
      Contact( #DataIn.Pos1_Ls )
      I_Contact( #DataIn.Pos0_Ls )
      I_Contact( #DataIn.Pos2_Ls )
      Move(in := 1, out1 => #COut.Paletto.Pos)
   END_RUNG
   RUNG wire#powerrail
      Contact( #DataIn.Pos2_Ls )
      I_Contact( #DataIn.Pos0_Ls )
      I_Contact( #DataIn.Pos1_Ls )
      Move(in := 2, out1 => #COut.Paletto.Pos)
   END_RUNG
   // the same network as SCL:
   #COut.Paletto.CtrlSafe := #V_1.COut.CtrlSafe OR #V_2.COut.CtrlSafe;
   #COut.Paletto.Standstill := #V_1.COut.Standstill AND #V_2.COut.Standstill;
   #COut.Paletto.Rest_CheckNext := #V_1.COut.Rest_CheckNext OR #V_2.COut.Rest_CheckNext;
   #COut.Paletto.Work_CheckNext := #V_1.COut.Work_CheckNext OR #V_2.COut.Work_CheckNext;
   #_w1 := #DataIn.Pos0_Ls AND NOT #DataIn.Pos1_Ls AND NOT #DataIn.Pos2_Ls;
   IF #_w1 THEN #COut.Paletto.Pos := 0; END_IF;
   #COut.Paletto.RestPosition := #_w1;
   IF #DataIn.Pos1_Ls AND NOT #DataIn.Pos0_Ls AND NOT #DataIn.Pos2_Ls THEN #COut.Paletto.Pos := 1; END_IF;
   IF #DataIn.Pos2_Ls AND NOT #DataIn.Pos0_Ls AND NOT #DataIn.Pos1_Ls THEN #COut.Paletto.Pos := 2; END_IF;
END_REGION

REGION Network 50: <<< MACHINE STATUS >>>
END_REGION

REGION Network 51: Collect machine to zone interface (internal machines OR)
   RUNG wire#powerrail
      "MachineInterface_2_To_1"(MachineInterface_1 := #Ax.MachineInterface, MachineInterface_2 := #V_1.MachineInterface, AdditionalAlarms := FALSE, AdditionalWarnings := FALSE, Ret_Val => #MachineInterface)
   END_RUNG
   RUNG wire#powerrail
      "MachineInterface_2_To_1"(AdditionalWarnings := wire#w1, MachineInterface_1 := #V_1.MachineInterface, MachineInterface_2 := #V_2.MachineInterface, AdditionalAlarms := FALSE, Ret_Val => #MachineInterface)
   END_RUNG
   RUNG wire#powerrail
      I_Contact( #Warning.MissingCnd.OP_REST )
      I_Contact( #Warning.MissingCnd.OP_WORK )
      I_Contact( #Warning.MissingCnd.AxInRestPos )
      Not()
   END_RUNG wire#w1
   // the same network as SCL:
   #MachineInterface := "MachineInterface_2_To_1"(MachineInterface_1 := #Ax.MachineInterface,
                           MachineInterface_2 := #V_1.MachineInterface,
                           AdditionalAlarms := FALSE,
                           AdditionalWarnings := FALSE);
   #MachineInterface := "MachineInterface_2_To_1"(MachineInterface_1 := #V_1.MachineInterface,
                           MachineInterface_2 := #V_2.MachineInterface,
                           AdditionalAlarms := FALSE,
                           AdditionalWarnings := NOT (NOT #Warning.MissingCnd.OP_REST AND NOT #Warning.MissingCnd.OP_WORK AND NOT #Warning.MissingCnd.AxInRestPos));
END_REGION
END_FUNCTION_BLOCK
